// TwinCAT 3 PLC project IPC
// Title: Modbus RTU Base
// Company: NewEngineer
// Author: https://github.com/phucpha
// ProjectVersion: 1.1.1.1
// Description: This Library is a use for Modbus Master and modbus Slave as Function block base for modbus RTU applications
// ProgramVersion: 3.1.4024.0
// libraries:
//   Tc2_ModbusRTU, * (Beckhoff Automation GmbH)
//   Tc2_Standard, * (Beckhoff Automation GmbH)
//   Tc3_Module, * (Beckhoff Automation GmbH)
// project tree:
//   DUTs/ E_ModbusFunction.TcDUT (not stored), E_ModBusMasterState.TcDUT, E_ModbusMasterStateRun.TcDUT
//   / PlcTask.TcTTO
//   POUs/ FB_ModbusMaster_PcCOM.TcPOU, FB_ModbusSlave.TcPOU, I_ModbusSlave.TcIO (not stored)
//   Version/ Global_Version.TcGVL
// real-time tasks:
//   TASK PlcTask: cycle T#10ms, priority 20, ADS port 350

CONFIGURATION IPC
    RESOURCE PLC ON TwinCAT3
        TASK PlcTask(INTERVAL := T#10ms, PRIORITY := 20);
    END_RESOURCE
END_CONFIGURATION

// ---- DUTs/E_ModBusMasterState.TcDUT
{attribute 'qualified_only'}
{attribute 'strict'}
TYPE E_ModBusMasterState :
(
	Uninitialized 	:= 0,
	Initializing 	:= 10,
	Ready			:= 20,
	Running			:= 30,
	Stop			:= 200,
	Stop_done		:= 210
	
);
END_TYPE

// ---- DUTs/E_ModbusMasterStateRun.TcDUT
{attribute 'qualified_only'}
{attribute 'strict'}
TYPE E_ModbusMasterStateRun :
(
	CheckNumberSlaveRegistered 	:= 0, 
	SetParametersRead 			:= 10,
	SendRequestRead				:= 20,
	WaitReadRespond				:= 40,
	ConvertRawData				:= 50,
	ReturnReadDone				:= 60,
	
	SetParametersWrite 			:= 70,
	SendRequestWrite			:= 80,
	WaitWriteRespond 			:= 90,
	ReturnWriteDone				:= 120
);
END_TYPE

// ---- Version/Global_Version.TcGVL
{attribute 'TcGenerated'}
{attribute 'no-analysis'}
{attribute 'linkalways'}
// This function has been automatically generated from the project information.
VAR_GLOBAL CONSTANT
	{attribute 'const_non_replaced'}
	stLibVersion_Modbus_RTU_Base : ST_LibVersion := (iMajor := 1, iMinor := 1, iBuild := 1, iRevision := 1, nFlags := 0, sVersion := '1.1.1.1');
END_VAR

// ---- POUs/FB_ModbusMaster_PcCOM.TcPOU
FUNCTION_BLOCK FB_ModbusMaster_PcCOM //IMPLEMENTS I_UniversalUnit
VAR
	sName			:		STRING;
	bInitialized	:		BOOL;
	iScantime		:		UINT := 50;
	iTimeout		:		UINT := 1000;//1000ms
	iErrorID		:		MODBUS_ERRORS;
	bBusy			: 		BOOL;
	bError			:		BOOL;
	iStepGeneral	: 		E_ModBusMasterState;
	iStepRunning	:		E_ModbusMasterStateRun;
	bFirstCycle		:		BOOL;
	bRun			:		BOOL;
	bStop			: 		BOOL;

	fbModbusMaster	: 		ModbusRtuMaster_PcCOM;
	ipModbusSlave	:		ARRAY [1..247] OF I_ModbusSlave;
	iAmountSlave	: 		UINT;
	
	iLoopSlave		:		UINT	:= 1;
	iLoopAdr		:		UINT;
	iQuantity 		: 		POINTER TO WORD;
	iMBAddr 		: 		POINTER TO WORD;
    arrData			: 		ARRAY [0..255] OF WORD;
	
	UnitId			: BYTE;
	Quantity		: WORD;
	MBAddr			: WORD;
	cbLength 		: UINT;
	pMemoryAddr		: POINTER TO BYTE;
	pDataWrite		: POINTER TO WORD;

	bexecute		: BOOL;
	
	tCalculateTimeRW	: TON;
	tTimerScanDelay		: TON;
	nNumberFaultRW		: UINT;
	eModbusFunction		: E_ModbusFunction;
	peModbusFunction 	: POINTER TO WORD;
END_VAR

StateMachine();
bRun :=  iStepGeneral = E_ModBusMasterState.Running ;
bStop := iStepGeneral = E_ModBusMasterState.stop_done;
bInitialized := iStepGeneral >= E_ModBusMasterState.Ready;
iErrorID := fbModbusMaster.ErrorId;

METHOD Abort : BOOL
bError := FALSE;
iErrorID := 0;
bError := FALSE;
iStepRunning	:= E_ModbusMasterStateRun.CheckNumberSlaveRegistered;
iLoopSlave		:= 1;
iLoopAdr		:= 0;
fbModbusMaster.WriteMultipleCoils( Execute := FALSE);
fbModbusMaster.WriteRegs( Execute := FALSE);
fbModbusMaster.WriteSingleCoil( Execute := FALSE);	
fbModbusMaster.WriteSingleRegister( Execute := FALSE);
fbModbusMaster.ReadRegs(Execute := FALSE);
fbModbusMaster.ReadInputRegs(Execute := FALSE);
IF NOT fbModbusMaster.BUSY THEN
	iStepGeneral	:= E_ModBusMasterState.Uninitialized;
	Abort := TRUE;
END_IF
END_METHOD

PROPERTY AnyError : BOOL
GET
AnyError 	:= bError;
END_GET
END_PROPERTY

PROPERTY Busy : BOOL
GET
Busy := bBusy;
END_GET
END_PROPERTY

PROPERTY CycleTimeMeasure : Time
GET
CycleTimeMeasure := tCalculateTimeRW.ET;
END_GET
END_PROPERTY

PROPERTY ErrorID : MODBUS_ERRORS
GET
ErrorID := iErrorID;
END_GET
END_PROPERTY

METHOD Init : BOOL
IF iStepGeneral = E_ModBusMasterState.Uninitialized THEN
	iStepGeneral := E_ModBusMasterState.Initializing;
END_IF

Init := (iStepGeneral >= E_ModBusMasterState.Ready);
END_METHOD

PROPERTY Initialized : BOOL
GET
Initialized := bInitialized;
END_GET
END_PROPERTY

PROPERTY Name : STRING
GET
Name := sName;
END_GET
SET
sName := Name;
END_SET
END_PROPERTY

PROPERTY ReadData : ARRAY [0..255] OF Word
GET
ReadData := arrData;
END_GET
END_PROPERTY

PROPERTY ReadDataSize : uint
GET
ReadDataSize := INT_TO_UINT(SIZEOF(arrData));
END_GET
END_PROPERTY

METHOD RegisterSlave : BOOL
VAR_INPUT
	ModbusSlave		:		I_ModbusSlave;
END_VAR
VAR
	iLoop	:	UINT;
	bExists	:	BOOL;
END_VAR
FOR iLoop := 1 TO iAmountSlave DO
	IF ipModbusSlave[iLoop] = ModbusSlave THEN
		bExists := TRUE;
		iLoop := iAmountSlave;// end loop for command
	END_IF
END_FOR 
IF NOT bExists THEN
	iAmountSlave := iAmountSlave + 1;
	ipModbusSlave[iAmountSlave] := ModbusSlave;
END_IF
END_METHOD

METHOD Reset : BOOL
bError := FALSE;
iErrorID := 0;
bError := FALSE;
iStepGeneral	:= E_ModBusMasterState.Uninitialized;
iStepRunning	:= E_ModbusMasterStateRun.CheckNumberSlaveRegistered;

iLoopSlave		:= 1;
iLoopAdr		:= 0;

fbModbusMaster.Execute := FALSE;

Reset := TRUE;
END_METHOD

METHOD Run : BOOL /// call from FB_modbus
IF (iStepGeneral = E_ModBusMasterState.Ready) THEN
	iStepGeneral := E_ModBusMasterState.Running;
END_IF

bRun := TRUE;
Run := (iStepGeneral >= E_ModBusMasterState.Running) AND (iStepGeneral < E_ModBusMasterState.stop);
END_METHOD

PROPERTY ScanTime : UINT
GET
ScanTime := iScantime;
END_GET
SET
iScantime := ScanTime;
END_SET
END_PROPERTY

METHOD protected StateInit : BOOL (*Unit is performing initialization*)
fbModbusMaster( Execute := FALSE,
	BUSY => bBusy,
	Error => bError,
	ErrorId => iErrorID
);
fbModbusMaster.ReadRegs(Execute := FALSE);
fbModbusMaster.ReadInputRegs(Execute := FALSE);
fbModbusMaster.WriteMultipleCoils( Execute := FALSE);
fbModbusMaster.WriteRegs( Execute := FALSE);
fbModbusMaster.WriteSingleCoil( Execute := FALSE);	
fbModbusMaster.WriteSingleRegister( Execute := FALSE);
IF NOT bError AND NOT bBusy THEN
	iStepGeneral := E_ModBusMasterState.Ready;
END_IF
END_METHOD

METHOD protected StateMachine : BOOL (*State machine of unit*)
CASE iStepGeneral OF
		E_ModBusMasterState.Uninitialized:  
			StateUninitialized();
	
		E_ModBusMasterState.Initializing: 
			StateInit();
	
		E_ModBusMasterState.Ready: 
			StateReady();
		
		E_ModBusMasterState.Running: 
			StateRunning();
						
		E_ModBusMasterState.stop:
			StateStopping();
			
		E_ModBusMasterState.stop_done:
			StateStoppingDone();
END_CASE
END_METHOD

METHOD protected StateReady : BOOL (* Unit is initialized*)
END_METHOD

METHOD PROTECTED StateRunning : BOOL (* Unit is uninitialized*)
VAR 
	

	
END_VAR
CASE iStepRunning OF
	E_ModbusMasterStateRun.CheckNumberSlaveRegistered: // Trigger
		tCalculateTimeRW(
			IN := TRUE,
			PT := T#5M
		);	
		IF iAmountSlave > 0 THEN
			iStepRunning := E_ModbusMasterStateRun.SetParametersRead;
		END_IF
			
	E_ModbusMasterStateRun.SetParametersRead: // Set parameters
		IF ipModbusSlave[iLoopSlave].NumAddRegionRead <> 0 
		AND iLoopAdr <= (ipModbusSlave[iLoopSlave].NumAddRegionRead - 1) 
		THEN
			iQuantity := ipModbusSlave[iLoopSlave].AddressRead + ((iLoopAdr * 3 + 1) * SIZEOF(WORD));// arrAddressRead[iloopAdr][1] in Slave
			iMBAddr := ipModbusSlave[iLoopSlave].AddressRead + ((iLoopAdr * 3) * SIZEOF(WORD));// arrAddressRead[iloopAdr][0] in Slave
			UnitID := ipModbusSlave[iLoopSlave].UnitID;
			Quantity :=	iQuantity^;
			MBAddr := iMBAddr^;
			cbLength := SIZEOF(arrData);
			pMemoryAddr	:= ADR(arrData);
			peModbusFunction := ipModbusSlave[iLoopSlave].AddressRead + ((iLoopAdr * 3 + 2) * SIZEOF(WORD)); // arrAddressRead[iloopAdr][2] in Slave
			eModbusFunction := peModbusFunction^;
			iStepRunning := E_ModbusMasterStateRun.SendRequestRead;
		ELSE 
			iLoopAdr := 0;
			iStepRunning := E_ModbusMasterStateRun.ReturnReadDone;
		END_IF

			
	E_ModbusMasterStateRun.SendRequestRead: // Send request
		CASE eModbusFunction OF
			E_ModbusFunction.ReadHoldingRegisters:
				fbModbusMaster.ReadRegs(
					UnitID:= UnitID, 
					Quantity:= Quantity, 
					MBAddr:= MBAddr, 
					cbLength:= cbLength, 
					pMemoryAddr:= pMemoryAddr, 
					Execute:= TRUE,
					Timeout:= UINT_TO_TIME(iTimeout),
					BUSY=> bBusy, 
					Error=> bError , 
					ErrorId=>iErrorId 
				);
			
			E_ModbusFunction.ReadInputRegisters:
				fbModbusMaster.ReadInputRegs(
					UnitID:= UnitID, 
					Quantity:= Quantity, 
					MBAddr:= MBAddr, 
					cbLength:= cbLength, 
					pMemoryAddr:= pMemoryAddr, 
					Execute:= TRUE,
					Timeout:= UINT_TO_TIME(iTimeout),
					BUSY=> bBusy, 
					Error=> bError , 
					ErrorId=>iErrorId 
				);
			
		END_CASE
		iStepRunning := E_ModbusMasterStateRun.WaitReadRespond;
						
	E_ModbusMasterStateRun.WaitReadRespond:
		fbModbusMaster.ReadRegs(Execute := FALSE);
		fbModbusMaster.ReadInputRegs(Execute := FALSE);
		IF NOT fbModbusMaster.BUSY AND NOT fbModbusMaster.Error THEN
			ipModbusSlave[iLoopSlave].ModbusErrorID := iErrorID;
			iStepRunning := E_ModbusMasterStateRun.ConvertRawData;
			nNumberFaultRW := 0;
		END_IF
		
		IF fbModbusMaster.Error AND NOT fbModbusMaster.BUSY THEN
			ipModbusSlave[iLoopSlave].ModbusErrorID := iErrorID;
			iStepRunning := E_ModbusMasterStateRun.ReturnReadDone;
		END_IF
	
	E_ModbusMasterStateRun.ConvertRawData: 
		ipModbusSlave[iLoopSlave].Convert(
			iRegionNo := iLoopAdr,
		 	pReadData := ADR(arrData)
		);
		iLoopAdr := iLoopAdr + 1;
		iStepRunning := E_ModbusMasterStateRun.CheckNumberSlaveRegistered;

	E_ModbusMasterStateRun.ReturnReadDone: // Return, done
		iStepRunning := E_ModbusMasterStateRun.SetParametersWrite;
		iLoopAdr := 0;

	E_ModbusMasterStateRun.SetParametersWrite :
		IF  ipModbusSlave[iLoopSlave].NumAddRegionWrite <> 0
		AND iLoopAdr <= ipModbusSlave[iLoopSlave].NumAddRegionWrite - 1 
		THEN // iLoopAdr start from 1
			iMBAddr := ipModbusSlave[iLoopSlave].AddressWrite + (iLoopAdr * 11 * SIZEOF(WORD));// return address word contain value address( modbus) 
			pDataWrite := ipModbusSlave[iLoopSlave].AddressWrite + ((iLoopAdr * 11 + 2) * SIZEOF(WORD));
			iQuantity := ipModbusSlave[iLoopSlave].AddressWrite + ((iLoopAdr * 11 + 1) * SIZEOF(WORD));
			peModbusFunction := ipModbusSlave[iLoopSlave].AddressWrite + ((iLoopAdr * 11 + 10) * SIZEOF(WORD));
			eModbusFunction := peModbusFunction^;
			UnitID 	:=		ipModbusSlave[iLoopSlave].UnitID;
			Quantity	:=	iQuantity^;
			MBAddr	:=		iMBAddr^;
			cbLength	:= 	Quantity * 2;
			pMemoryAddr	:= 	pDataWrite;
			iStepRunning := E_ModbusMasterStateRun.SendRequestWrite;
		ELSE 
			iStepRunning := E_ModbusMasterStateRun.ReturnWriteDone;
		END_IF

	E_ModbusMasterStateRun.SendRequestWrite :
		CASE eModbusFunction OF
			E_ModbusFunction.WriteMultipleCoils:
				fbModbusMaster.WriteMultipleCoils(
					UnitID:= UnitID, 
					Quantity:= Quantity, 
					MBAddr:= MBAddr, 
					cbLength:= cbLength, 
					pMemoryAddr:= pMemoryAddr, 
					Execute:=  true,
					Timeout:= 	UINT_TO_TIME(iTimeout),	
					BUSY=> bBusy, 
					Error=> bError , 
					ErrorId=>iErrorId 
				);
													
			E_ModbusFunction.WriteMultipleRegisters:
				fbModbusMaster.WriteRegs(
					UnitID:= UnitID, 
					Quantity:= Quantity, 
					MBAddr:= MBAddr, 
					cbLength:= cbLength, 
					pMemoryAddr:= pMemoryAddr, 
					Execute:= TRUE,
					Timeout:= UINT_TO_TIME(iTimeout),	
					BUSY=> bBusy, 
					Error=> bError , 
					ErrorId=>iErrorId 
				);
											
			E_ModbusFunction.WriteSingleCoil:
				fbModbusMaster.WriteSingleCoil(
					UnitID:= UnitID, 
					Quantity:= Quantity, 
					MBAddr:= MBAddr, 
					cbLength:= cbLength, 
					pMemoryAddr:= pMemoryAddr, 
					Execute:=  true,
					Timeout:= UINT_TO_TIME(iTimeout),	
					BUSY=> bBusy, 
					Error=> bError , 
					ErrorId=>iErrorId 
				);
			E_ModbusFunction.WriteSingleRegister:
				fbModbusMaster.WriteSingleRegister(
					UnitID:= UnitID, 
					Quantity:= Quantity, 
					MBAddr:= MBAddr, 
					cbLength:= cbLength, 
					pMemoryAddr:= pMemoryAddr, 
					Execute:=  true,
					Timeout:= 	UINT_TO_TIME(iTimeout),	
					BUSY=> bBusy, 
					Error=> bError , 
					ErrorId=>iErrorId 
				);
		END_CASE
		
		iStepRunning := E_ModbusMasterStateRun.WaitWriteRespond;
	
	E_ModbusMasterStateRun.WaitWriteRespond :
		fbModbusMaster.WriteMultipleCoils( Execute := FALSE);
		fbModbusMaster.WriteRegs( Execute := FALSE);
		fbModbusMaster.WriteSingleCoil( Execute := FALSE);	
		fbModbusMaster.WriteSingleRegister( Execute := FALSE);
		IF NOT fbModbusMaster.BUSY AND NOT fbModbusMaster.Error THEN
			ipModbusSlave[iLoopSlave].ModbusErrorID := iErrorID;
			iStepRunning := E_ModbusMasterStateRun.SetParametersWrite;
			nNumberFaultRW := 0;
			iLoopAdr := iLoopAdr + 1;
		END_IF
		IF fbModbusMaster.Error AND NOT fbModbusMaster.BUSY THEN
			ipModbusSlave[iLoopSlave].ModbusErrorID := iErrorID;
			iStepRunning := E_ModbusMasterStateRun.ReturnWriteDone ;
		END_IF
	
	 E_ModbusMasterStateRun.ReturnWriteDone :
		iLoopAdr := 0;
		iLoopSlave := iLoopSlave + 1;// next slave
		IF iLoopSlave > iAmountSlave THEN
			iLoopSlave := 1;
		END_IF
		tTimerScanDelay( 
			IN := TRUE,
			PT := UINT_TO_TIME(iScantime)
		);
		IF tTimerScanDelay.Q THEN
			tTimerScanDelay( IN := FALSE);
			tCalculateTimeRW(in := FALSE);
		 	iStepRunning := E_ModbusMasterStateRun.CheckNumberSlaveRegistered;
		END_IF
			
END_CASE
END_METHOD

METHOD protected StateStopping : BOOL (* Unit is uninitialized*)
iStepRunning	:= E_ModbusMasterStateRun.CheckNumberSlaveRegistered;
iLoopSlave		:= 1;
iLoopAdr		:= 0;
fbModbusMaster.WriteMultipleCoils( Execute := FALSE);
fbModbusMaster.WriteRegs( Execute := FALSE);
fbModbusMaster.WriteSingleCoil( Execute := FALSE);	
fbModbusMaster.WriteSingleRegister( Execute := FALSE);
fbModbusMaster.ReadRegs(Execute := FALSE);
fbModbusMaster.ReadInputRegs(Execute := FALSE);
IF NOT fbModbusMaster.BUSY THEN
 	iStepGeneral := E_ModBusMasterState.Stop_done;
END_IF
END_METHOD

METHOD protected StateStoppingDone : BOOL (* Unit is uninitialized*)
IF NOT bStop THEN
	iStepGeneral := E_ModBusMasterState.Ready;
END_IF
END_METHOD

METHOD protected StateUninitialized : BOOL (* Unit is uninitialized*)
END_METHOD

METHOD protected Stop : BOOL
IF iStepGeneral >= E_ModBusMasterState.Running AND iStepGeneral < E_ModBusMasterState.stop THEN
	iStepGeneral := E_ModBusMasterState.stop;
END_IF
bStop := TRUE;

Stop := (iStepGeneral = E_ModBusMasterState.stop_done);
END_METHOD

PROPERTY Stopped : bool
GET
Stopped := bStop;
END_GET
END_PROPERTY

PROPERTY Timeout : UINT // in milisecond, if not respond in this time , error will raise
GET
Timeout := iTimeout;
END_GET
SET
iTimeout := Timeout;
END_SET
END_PROPERTY

END_FUNCTION_BLOCK

// ---- POUs/FB_ModbusSlave.TcPOU
FUNCTION_BLOCK FB_ModbusSlave IMPLEMENTS I_ModbusSlave
VAR
	iUnitID	:	BYTE; // address of the Slave
	arrAddressRead	:	ARRAY [0..50] OF ARRAY [0..2] OF WORD;
	(*arrAddressRead[x][y]: +x : index of Region Read.  arrAddressRead[0]: the first region Read.
							+y:
								case y of
									0: Register address for Read
									1: Number of register for read
									2: Function Read
					 *)
	iNumAddRegionRead	:	UINT;
	
	arrAddressWrite		: ARRAY [0..20] OF ARRAY [0..10] OF WORD;// write Multiple or single register
	(* the 20 is max number of region write,
		arrAddressWrite[x][y] : +x: index of Region Read.  arrAddressRead[0]: the first region Read. 
								+y:
									case y of
										0 :  Register address for Write
										1 : number of register will be write => modbus master automatic choose Function Write( single Register or Multi Regiseter)
										2..9 : max 8 value for write
										10: Write Function : e.g E_ModbusFunction.WriteSingleCoil
															
	*)
	iNumAddRegionWrite	: UINT;
	sName				:		STRING;
	bFirstCycle 		: 		BOOL := TRUE;
	iModbusErrorID		:		MODBUS_ERRORS;
END_VAR

PROPERTY AddressRead : POINTER TO WORD
GET
AddressRead := ADR(arrAddressRead);
END_GET
END_PROPERTY

PROPERTY AddressWrite : POINTER TO WORD
GET
AddressWrite := ADR( arrAddressWrite);
END_GET
END_PROPERTY

METHOD Convert : BOOL
VAR_INPUT
	iRegionNo	:	INT;
	pReadData	:	POINTER TO word;
END_VAR
END_METHOD

METHOD FirstCycle // must be call once time 
VAR_INPUT
	sName : STRING;
	iUnitID : BYTE ; // modbus address of the device : 1- 255
END_VAR
THIS^.sName := sName;
THIS^.iUnitID := iUnitID;
END_METHOD

{attribute 'monitoring' := 'variable'}
PROPERTY ModbusErrorID : MODBUS_ERRORS
GET
ModbusErrorID := iModbusErrorID;
END_GET
SET
iModbusErrorID := ModbusErrorID;
END_SET
END_PROPERTY

PROPERTY Name : STRING
GET
Name := sName;
END_GET
SET
sName := Name;
END_SET
END_PROPERTY

PROPERTY NumAddRegionRead : UINT
GET
NumAddRegionRead := iNumAddRegionRead;
END_GET
END_PROPERTY

PROPERTY NumAddRegionWrite : UINT
GET
NumAddRegionWrite := iNumAddRegionWrite;
END_GET
END_PROPERTY

PROPERTY UnitID : BYTE
GET
UnitID := iUnitID;
END_GET
SET
iUnitID := UnitID;
END_SET
END_PROPERTY

END_FUNCTION_BLOCK
